TYPE EL5042_Data :
STRUCT
	{attribute addProperty Name "FB Inputs Channel 1"}
	FB_InputsChannel_1 : EL5032_FB_InputsChannel;
	{attribute addProperty Name "FB Inputs Channel 2"}
	FB_InputsChannel_2 : EL5032_FB_InputsChannel;
END_STRUCT
END_TYPE

(* stored: Version 1.1.0.1, ProductVersion 3.1.4024.9
   DUT EL5042_Data: Id {bfe94409-e5c5-0644-3ac5-74814ff4eda5} *)
